// TIA Portal V20 export
DATA_BLOCK "FB_FlowMeter_DB_2"   // DB4
// stored: InstanceOfName FB_FlowMeter_FDH32, InstanceOfType FB
"FB_FlowMeter_FDH32"
   // VAR_INPUT
   //    iUnscaled_Min : Real;
   //    iUnscaled_Max : Real;
   //    iScaled_Flow_Min : Real;
   //    iFlow_Raw : Int;
   //    iQuittieren : Bool;
   //    iImpuls : Bool;
   //    iStoerungUnterdr : Bool;
   //    iPipe_diameter : Bool;
   //    iMin_FlowRate : Real;
   //    iMax_FlowRate : Real;
   //    iTemp_Raw : Word;
   //    iScaled_Temp_Min : Real;
   //    iScaled_Temp_Max : Real;
   //    iTemp_Above_Limit { ExternalAccessible := 'False'; ExternalVisible := 'False'; ExternalWritable := 'False'} : Real;
   //    iTemp_Below_limit : Real;
   //    iErrorFrom_Sensor : Bool;
   //    iAssembly_Place : String;
   // END_VAR
   // VAR_OUTPUT
   //    oOutSteo : "UDT_Flowmeter_Stoe";
   // END_VAR
   // VAR_IN_OUT
   //    ioVisuSteuern : "UDT_Flowmeter_Steuern";
   //    ioVisuStatus : "UDT_Flowmeter_Status";
   // END_VAR
   // VAR
   //    sFlow_ScaledValue : Real;
   //    sTemp_ScaledValue : Real;
   //    Buffer : Array[1..10] of Real;
   //    Index : DInt;
   //    Sum : Real;
   //    sScaled_Max : Real;
   //    i : Int;
   //    sAvg : Real;
   //    sCyclecount : Real;
   //    sOut_I : Int;
   // END_VAR
BEGIN
END_DATA_BLOCK
